// TwinCAT 3 PLC project PLC
// ProgramVersion: 3.1.4024.0
// libraries:
//   SPT Base Types, * (Beckhoff Automation LLC)
//   SPT Components, * (Beckhoff Automation LLC)
//   SPT Diagnostic, * (Beckhoff Automation LLC)
//   SPT EtherCat, * (Beckhoff Automation LLC)
//   SPT Event Logger, * (Beckhoff Automation LLC)
//   SPT Kinematics, * (Beckhoff Automation LLC)
//   SPT Motion Control, * (Beckhoff Automation LLC)
//   SPT NCI, * (Beckhoff Automation LLC)
//   SPT Utilities, * (Beckhoff Automation LLC)
//   SPT Vision, * (Beckhoff Automation LLC)
//   SPT XTS, * (Beckhoff Automation LLC)
//   Tc2_MC2, * (Beckhoff Automation GmbH)
//   Tc2_Standard, * (Beckhoff Automation GmbH)
//   Tc2_System, * (Beckhoff Automation GmbH)
//   Tc3_EventLogger, * (Beckhoff Automation GmbH)
//   Tc3_Module, * (Beckhoff Automation GmbH)
//   Tc3_PackML_V2, * (Beckhoff Automation GmbH)
// project tree:
//   / FastTask.TcTTO, GlobalTextList.TcGTLO, PlcTask.TcTTO, Visualization Manager.TcVMO (not stored)
//   Function Blocks/ExternalSetpointGenerator/ E_ExternalSPGen.TcDUT, FB_ExternalSetpointGenerator.TcPOU, I_ExternalSetpointGenerator.TcIO
//   Modules/00 Machine/ Machine.TcPOU
//   Modules/01 Infeed Position/ Infeed.TcPOU
//   Modules/02 Outfeed Velocity/ Outfeed.TcPOU
//   POUs Fast Task/ BasicESPG_Position.TcPOU, BasicESPG_Velocity.TcPOU, Fast_Task.TcPOU
//   POUs/ MAIN.TcPOU
//   VISUs/ Visualization.TcVIS, Basic_ESPG.TcVIS
// real-time tasks:
//   TASK PlcTask: cycle T#10ms, priority 20, ADS port 350
//   TASK FastTask: cycle T#2ms, priority 1, ADS port 351
// motion (NC):
//   TASK NC-Task 1 SAF: cycle T#2ms, priority 4, ADS port 501
//   TASK NC-Task 1 SVB: cycle T#10ms, priority 8, ADS port 511
//   AXIS Axis Position (id 1)
//     OtherSettings: AllowMotionCmdToSlave=true
//     encoder EncType=1
//     drive DrvType=5
//       Analog: TorqueSetpointScale=10, ScaleFactorActTorque=0.1
//       TimeComp: TaskDelayCycles=1
//     controller CtrType=1
//       CtrPara: PriorControlFactor=1
//         Observer: BandWidth=20
//   AXIS Axis Velocity (id 4)
//     OtherSettings: AllowMotionCmdToSlave=true
//     encoder EncType=1
//     drive DrvType=5
//       Analog: TorqueSetpointScale=10, ScaleFactorActTorque=0.1
//       TimeComp: TaskDelayCycles=1
//     controller CtrType=1
//       CtrPara: PriorControlFactor=1
//         Observer: BandWidth=20
//   AXIS Basic ESPG Velocity (id 3)
//   AXIS Basic ESPG Position (id 2)
// variable links:
//   PLC/PLC Instance <-> NC-Task 1 SAF/Axes/Axis Position
//     FastTask Inputs/Fast_Task.PositionAxis.BasicAxis._Axis.NcToPlc <-> Outputs/ToPlc
//     FastTask Outputs/Fast_Task.PositionAxis.BasicAxis._Axis.PlcToNc <-> Inputs/FromPlc
//   PLC/PLC Instance <-> NC-Task 1 SAF/Axes/Axis Velocity
//     FastTask Inputs/Fast_Task.VelocityAxis.BasicAxis._Axis.NcToPlc <-> Outputs/ToPlc
//     FastTask Outputs/Fast_Task.VelocityAxis.BasicAxis._Axis.PlcToNc <-> Inputs/FromPlc
//   PLC/PLC Instance <-> NC-Task 1 SAF/Axes/Basic ESPG Position
//     FastTask Inputs/BasicESPG_Position.Basic_Axis.NcToPlc <-> Outputs/ToPlc
//     FastTask Outputs/BasicESPG_Position.Basic_Axis.PlcToNc <-> Inputs/FromPlc
//   PLC/PLC Instance <-> NC-Task 1 SAF/Axes/Basic ESPG Velocity
//     FastTask Inputs/BasicESPG_Velocity.Basic_Axis.NcToPlc <-> Outputs/ToPlc
//     FastTask Outputs/BasicESPG_Velocity.Basic_Axis.PlcToNc <-> Inputs/FromPlc

CONFIGURATION PLC
    RESOURCE PLC ON TwinCAT3
        TASK FastTask(INTERVAL := T#2ms, PRIORITY := 1);
        TASK PlcTask(INTERVAL := T#10ms, PRIORITY := 20);
        PROGRAM Fast_Task WITH FastTask : Fast_Task;
        PROGRAM MAIN WITH PlcTask : MAIN;
    END_RESOURCE
END_CONFIGURATION

// ---- Function Blocks/ExternalSetpointGenerator/E_ExternalSPGen.TcDUT
{attribute 'qualified_only'}
{attribute 'strict'}
TYPE E_ExternalSPGen : (
		Wait := 0,
		EnableCmd,
		Enabling,
		Feeding,
		DisableCmd,
		Disabling,
		Error
	);
END_TYPE

// ---- Function Blocks/ExternalSetpointGenerator/I_ExternalSetpointGenerator.TcIO
INTERFACE I_ExternalSetpointGenerator

PROPERTY Accel : lreal
GET
END_GET
SET
END_SET
END_PROPERTY

PROPERTY Destination : lreal
GET
END_GET
SET
END_SET
END_PROPERTY

PROPERTY Direction : DINT // -1 = negative direction, 0 = standstill, 1 = positive direction
GET
END_GET
SET
END_SET
END_PROPERTY

METHOD Disable : bool
VAR_INPUT
END_VAR
END_METHOD

PROPERTY Position : lreal
GET
END_GET
SET
END_SET
END_PROPERTY

PROPERTY Velocity : lreal
GET
END_GET
SET
END_SET
END_PROPERTY

END_INTERFACE

// ---- POUs Fast Task/Fast_Task.TcPOU
PROGRAM Fast_Task
VAR
	PositionAxis	  : FB_Component_BasicAxis := (Name := 'Position Axis');
	PosExtSetpointGen : FB_ExternalSetpointGenerator;
	VelocityAxis	  : FB_Component_BasicAxis := (Name := 'Velocity Axis');
	VelExtSetpointGen : FB_ExternalSetpointGenerator;
END_VAR

(*
	External Setpoint Generator
	This code is the standard implementation of the External Setpoint Generator
	Use this along with the Bassic_ESPG Visu to become familiar with how it works if you have not used the External Setpoint Generator before
	This code is not used by the SPT Framework Implmentation
*)
BasicESPG_Position();
BasicESPG_Velocity();

(*****************************************************************************************************************************************************************)

(*****************************************************************************************************************************************************************)

(*****************************************************************************************************************************************************************)

(*
	These components are defined in this fast task in order for the values of the External Setpoint Generator
	to be updated and transfered to the motion controler at the speed of the fast task.
	These components are controlled and monitored through their interfaces from an EM 
*)

// Infeed EM
PositionAxis.CyclicLogic();
PositionAxis.ExternalSequence := PosExtSetpointGen;

//Outfeed EM
VelocityAxis.CyclicLogic();
VelocityAxis.ExternalSequence := VelExtSetpointGen;

END_PROGRAM

// ---- Function Blocks/ExternalSetpointGenerator/FB_ExternalSetpointGenerator.TcPOU
FUNCTION_BLOCK FB_ExternalSetpointGenerator EXTENDS FB_CyclicFB IMPLEMENTS I_MotionSequence, I_ExternalSetpointGenerator
VAR
	//Properties
	_Axis		 : I_BasicAxis;
	_Position	 : LREAL;
	_Destination : LREAL := 0.0;
	_Velocity	 : LREAL := 0.0;
	_Accel		 : LREAL := 0.0;
	_Direction	 : DINT	 := 1;

	// FBs
	EnableExtSP	 : MC_ExtSetPointGenEnable;
	DisableExtSP : MC_ExtSetPointGenDisable;

	//Internal Vars
	SequenceStep : INT;
	Options		 : ST_ExtSetPointEnableOptions;
END_VAR

PROPERTY Accel : lreal
GET
Accel := _Accel;
END_GET
SET
_Accel := Accel;
END_SET
END_PROPERTY

{warning 'add property implementation'}
PROPERTY Axis : SPT_Motion_Control.I_BasicAxis
GET
Axis := _Axis;
END_GET
SET
_Axis := Axis;
END_SET
END_PROPERTY

{warning 'add method implementation '}
METHOD CyclicLogic

VAR
	_Pos		 : LREAL;
END_VAR
CASE SequenceStep OF
	E_ExternalSPGen.Wait:
		EnableExtSP(Axis := _Axis.Axis, Execute := FALSE, Position := _Axis.ActualPosition);
		DisableExtSP(Axis := _Axis.Axis, Execute := FALSE);

	E_ExternalSPGen.EnableCmd:
		EnableExtSP(Axis		 := _Axis.Axis,
					Execute		 := TRUE,
					Position	 := _Destination, // Used for Position Monitoring
					PositionType := E_PositionType.POSITIONTYPE_ABSOLUTE,
					Options		 := Options);

		IF EnableExtSP.Enabled THEN
			SequenceStep := E_ExternalSPGen.Feeding;
		END_IF

	E_ExternalSPGen.Feeding:
		MC_ExtSetPointGenFeed(Axis		   := _Axis.Axis,
							  Position	   := _Position,
							  Velocity	   := _Velocity,
							  Acceleration := _Accel,
							  Direction	   := _Direction);

	E_ExternalSPGen.DisableCmd:
		DisableExtSP(Axis := _Axis.Axis, Execute := TRUE);
		SequenceStep := E_ExternalSPGen.Disabling;

	E_ExternalSPGen.Disabling:
		DisableExtSP(Axis := _Axis.Axis, Execute := FALSE);
		IF NOT DisableExtSP.Busy AND NOT DisableExtSP.Enabled THEN
			IF NOT DisableExtSP.Error THEN
				SequenceStep := E_ExternalSPGen.Wait;
			ELSE
				_ErrorID	 := DisableExtSP.ErrorID;
				SequenceStep := E_ExternalSPGen.Error;
			END_IF
		END_IF

	E_ExternalSPGen.Error:
		_Error := TRUE;
END_CASE

IF _Axis.Error THEN
	SequenceStep := E_ExternalSPGen.DisableCmd;
END_IF

//
_Busy := (SequenceStep <> 0) AND (NOT _Axis.Error);
END_METHOD

PROPERTY Destination : lreal
GET
Destination := _Destination;
END_GET
SET
_Destination := Destination;
END_SET
END_PROPERTY

PROPERTY Direction : DINT // -1 = negative direction, 0 = standstill, 1 = positive direction
GET
Direction := _Direction;
END_GET
SET
_Direction := Direction;
END_SET
END_PROPERTY

METHOD Disable : bool
VAR_INPUT
END_VAR
IF (_Axis = 0) THEN
	RETURN;
END_IF

_Busy		 := TRUE;
_Error		 := FALSE;
_ErrorID	 := 0;
SequenceStep := E_ExternalSPGen.DisableCmd;
Disable		 := TRUE;
END_METHOD

{warning 'add method implementation '}
METHOD Execute : BOOL
IF (_Axis = 0) OR _Busy THEN
	RETURN;
END_IF

_Busy		 := TRUE;
_Error		 := FALSE;
_ErrorID	 := 0;
SequenceStep := E_ExternalSPGen.EnableCmd;
Execute		 := TRUE;
END_METHOD

PROPERTY Position : lreal
GET
Position := _Position;
END_GET
SET
_Position := Position;
END_SET
END_PROPERTY

PROPERTY Velocity : lreal
GET
Velocity := _Velocity;
END_GET
SET
_Velocity := Velocity;
END_SET
END_PROPERTY

END_FUNCTION_BLOCK

// ---- POUs Fast Task/BasicESPG_Position.TcPOU
PROGRAM BasicESPG_Position
VAR
	Basic_Axis : AXIS_REF;
	Power	   : MC_Power;
	EnableSPG  : MC_ExtSetPointGenEnable;
	DisableSPG : MC_ExtSetPointGenDisable;

	//
	Execute					: BOOL;
	Destination				: LREAL;
	NextIncrementalPosition : LREAL;
	
	Inc1: BOOL;
	Inc10: BOOL;
	Dec1: BOOL;
	Dec10: BOOL;
	HasJob: BOOL;
END_VAR

// The Axis is always enabled for demo purposes
Power(Axis			  := Basic_Axis,
	  Enable		  := TRUE,
	  Enable_Positive := TRUE,
	  Enable_Negative := TRUE);

(*
	Enable the External Setpoint Generator and set the Destination
	The Destination value is loaded when the ESPG is ENabled
	This value will be used to determine the 'In Target Pos' and 'In Pos Range' flags
*)
EnableSPG(Axis := Basic_Axis, Execute := Execute, Position := Destination);

// Disable the External Setpoint Generator when not enabled
DisableSPG(Axis := Basic_Axis, Execute := NOT Execute);

(*
	Once enabled above, the Position value can be modified to send commands to the axis through the Axis.PlcToNc.ExtSetPos
	Velocity is not required as the MC_ExtSetPointGenFeed is sending position commands to the axis 
	- Actualy velocity for a real axis will be based on encoder feedback
	- For a simulation axis, actual velocity will be calculated based on the change in position and the task time
	An Acceleration value is not required for Position commands
	If the Direction is 0 the axis will not move, set the value to 1 for movemnt. The actual direction will be determined by the change in Position
*)

// When the Axis Status 'Has Job' is true, no other commands can be sent to the Axis. While the ESPG is Enabled, the 'Has Job' will be TRUE 
HasJob := Basic_Axis.NcToPlc.StateDWord.8;

//
IF EnableSPG.Enabled THEN // Not required, but prevents the NextIncrementalPosition value from being sent to Axis.PlcToNc.ExtSetPos
	MC_ExtSetPointGenFeed(Axis		   := Basic_Axis,
						  Position	   := NextIncrementalPosition,
						  Velocity	   := 0,
						  Acceleration := 0,
						  Direction	   := 1);
END_IF

(*	WARNING !!!!!!!!
	Changing the Position while the ESPG is not Enabled will change the value of the Axis.PlcToNc.ExtSetPos, but will not cause Axis movement.
	Enabling the ESPG with a Position value that is different than the current Actual Value will cause the axis to jump and likely fault.
*)

// Commands from Visu
IF Inc1 THEN
	Inc1					:= FALSE;
	NextIncrementalPosition := NextIncrementalPosition + 1;
END_IF

IF Inc10 THEN
	Inc10					:= FALSE;
	NextIncrementalPosition := NextIncrementalPosition + 10;
END_IF

IF Dec1 THEN
	Dec1					:= FALSE;
	NextIncrementalPosition := NextIncrementalPosition - 1;
END_IF

IF Dec10 THEN
	Dec10					:= FALSE;
	NextIncrementalPosition := NextIncrementalPosition - 10;
END_IF

END_PROGRAM

// ---- POUs Fast Task/BasicESPG_Velocity.TcPOU
PROGRAM BasicESPG_Velocity
VAR
	Basic_Axis : AXIS_REF;
	Power	   : MC_Power;
	EnableSPG  : MC_ExtSetPointGenEnable;
	DisableSPG : MC_ExtSetPointGenDisable;

	//
	Execute					: BOOL;
	NextIncrementalVelocity : LREAL;
	
	Inc1: BOOL;
	Inc10: BOOL;
	Dec1: BOOL;
	Dec10: BOOL;
	HasJob: BOOL;
END_VAR

// The Axis is always enabled for demo purposes
Power(Axis			  := Basic_Axis,
	  Enable		  := TRUE,
	  Enable_Positive := TRUE,
	  Enable_Negative := TRUE);

// Enable the External Setpoint Generator
EnableSPG(Axis := Basic_Axis, Execute := Execute, Position := 0);

// Disable the External Setpoint Generator when not enabled
DisableSPG(Axis := Basic_Axis, Execute := NOT Execute);

(*
	Once enabled above, the Velocity value can be modified to send commands to the axis through the Axis.PlcToNc.ExtSetVelo
	Position is not required as the MC_ExtSetPointGenFeed is sending Velocity commands to the axis 
	- Actualy velocity for a real axis will be based on encoder feedback
	- For a simulation axis, actual velocity will be 0 and the Actual Position will not change
	An Acceleration value is not required for Velocity commands
	If the Direction is 0 the axis will not move, set the value to 1 for movemnt. The actual direction will be determined by the sign of the Velocity
*)

// When the Axis Status 'Has Job' is true, no other commands can be sent to the Axis. While the ESPG is Enabled, the 'Has Job' will be TRUE 
HasJob := Basic_Axis.NcToPlc.StateDWord.8;

//
IF EnableSPG.Enabled THEN // Not required, but prevents the NextIncrementalVelocity value from being sent to Axis.PlcToNc.ExtSetVelo
	MC_ExtSetPointGenFeed(Axis		   := Basic_Axis,
						  Position	   := 0,
						  Velocity	   := NextIncrementalVelocity,
						  Acceleration := 0,
						  Direction	   := 1);
END_IF

(*	WARNING !!!!!!!!
	Changing the Velocity while the ESPG is not Enabled will change the value of the Axis.PlcToNc.ExtSetVelo, but will not cause Axis movement.
*)

// Commands from Visu
IF Inc1 THEN
	Inc1					:= FALSE;
	NextIncrementalVelocity := NextIncrementalVelocity + 1;
END_IF

IF Inc10 THEN
	Inc10					:= FALSE;
	NextIncrementalVelocity := NextIncrementalVelocity + 10;
END_IF

IF Dec1 THEN
	Dec1					:= FALSE;
	NextIncrementalVelocity := NextIncrementalVelocity - 1;
END_IF

IF Dec10 THEN
	Dec10					:= FALSE;
	NextIncrementalVelocity := NextIncrementalVelocity - 10;
END_IF

END_PROGRAM

// ---- POUs/MAIN.TcPOU
PROGRAM MAIN
VAR
	Machine : Machine := (Name := 'Machine');
END_VAR

(*All sample code provided by Beckhoff Automation LLC are for illustrative purposes only and are provided “as is” and without any warranties, express or implied. Actual implementations in applications will vary significantly. Beckhoff Automation LLC shall have no liability for, and does not waive any rights in relation to, any code samples that it provides or the use of such code samples for any purpose.*)

// NOTE: This code has not been tested on Hardware

// This is for debug only and should be removed
_AppInfo.KeepOutputsOnBP := TRUE;

(*
	There are 2 Equipment modules that use 1 axis each
	The Infeed EM controls an axis that implements Position control
	The Outfeed EM controls an axis that implements Velocity control
	
	Because the External Setpoint Generator provides smoother performce in a faster task,
	the Axis Components are defined within a POU that is updated by a 2ms Fast_Task.

	The fast task only calls the cyclic logic of the components, and sets the External Sequence of the component to the External Setpoint Generator.
	The EMs defined under the Machine Module have an interface that is assigned to the components in the Fast_Task.
	Through this interface the EM can control the component as if it was defined locally.
*)
Machine.CyclicLogic();

END_PROGRAM

// ---- Modules/00 Machine/Machine.TcPOU
FUNCTION_BLOCK Machine EXTENDS FB_PackML_BaseModule
VAR
	Infeed	: Infeed  := (Name := 'Infeed');
	Outfeed : Outfeed := (Name := 'Outfeed');
END_VAR

// Automatically enables and disables HMI control based on the PackML mode
METHOD PROTECTED HMIPermissions

// This method is called cyclically by CyclicLogic()
AllowHMIControl(TRUE);
END_METHOD

// Basic module initialization logic
METHOD PROTECTED Initialize : BOOL;
VAR
END_VAR

// This method is called by CyclicLogic() as required
Initialize := FALSE;
CASE DescendantSequenceState OF
	0:
		RegisterSubmodule(SubModule := Infeed);
		RegisterSubmodule(SubModule := Outfeed);
		DescendantSequenceState := DescendantSequenceState + 10;

	10:
		IF SUPER^.Initialize() THEN
			DescendantSequenceState := DescendantSequenceState + 10;
		END_IF

	20:
		Initialize := TRUE;
END_CASE
END_METHOD

END_FUNCTION_BLOCK

// ---- Modules/01 Infeed Position/Infeed.TcPOU
FUNCTION_BLOCK Infeed EXTENDS FB_PackML_BaseModule
VAR
	iInfeedxis				   : I_BasicAxis;				  // For most axis and component commands
	iInfeedAxisComponent	   : I_ComponentBase;			  // For registering the component with the EM
	iExternalSetpointGenerator : I_ExternalSetpointGenerator; // For setting properties of the External Setpoint Generator
END_VAR

// This method contains code which will execute when this PackML module is in the Aborting state
METHOD PROTECTED Aborting
VAR
	i				: UDINT;
	SubModulesReady : BOOL := TRUE;
END_VAR

// Note: The Abort command should be associated with the fault handing routine of a module. It should not be directly commanded from any user inteface. 

// This method is called as required by <c>StateControl()</c>
CASE SequenceState OF
	0:
		NoStateTasksToComplete := FALSE;
		SequenceState		   := SequenceState + 10;

	10:
		IF NOT iInfeedxis.Error THEN
			IF iInfeedxis.Stop() THEN
				SequenceState := SequenceState + 10;
			END_IF
		ELSE
			SequenceState := SequenceState + 10;
		END_IF

	20:
		IF iInfeedxis.Stopped THEN
			SequenceState := SequenceState + 10;
		END_IF

	30:
		IF iInfeedxis.Disable() THEN
			SequenceState := SequenceState + 10;
		END_IF

	40:
		IF NOT iInfeedxis.Enabled THEN
			SequenceState := SequenceState + 10;
		END_IF

	50:
		StateTasksComplete := TRUE;
END_CASE

SUPER^.Aborting();
END_METHOD

// This method contains code which will execute when this PackML module is in the Clearing state
METHOD PROTECTED Clearing
VAR
	i				: UDINT;
	SubModulesReady : BOOL := TRUE;
END_VAR

// Note: The Clear command can also be thought of as a fault reset depite the ambiguity in the naming of the Reset state. 

// This method is called as required by <c>StateControl()</c>
CASE SequenceState OF
	0:
		NoStateTasksToComplete := FALSE;
		SequenceState		   := SequenceState + 10;

	10:
		IF iInfeedxis.Reset() THEN
			SequenceState := SequenceState + 10;
		END_IF

	20:
		IF NOT iInfeedxis.Error THEN
			SequenceState := SequenceState + 10;
		END_IF

	30:
		StateTasksComplete := TRUE;
END_CASE

SUPER^.Clearing();
END_METHOD

// This method contains code which will execute when this PackML module is in the Execute state
METHOD PROTECTED Execute

(*
The base implementation of this method is empty. User must override this method to provide functionality.
This method is called as required by StateControl()
*)

VAR
	Position: LREAL;
END_VAR
CASE _CurrentMode OF
	E_PMLUnitMode.ePMLUnitMode_Production:
		CASE SequenceState OF
			0:
				iExternalSetpointGenerator.Direction   := 1;
				iExternalSetpointGenerator.Destination := 100.0;
				iExternalSetpointGenerator.Velocity	   := 0.0;
				iExternalSetpointGenerator.Accel	   := 0.0;
				SequenceState						   := 10;

			10:
				IF iInfeedxis.RunExternalSequence() THEN
					SequenceState := 20;
				END_IF

			20:
				IF iInfeedxis.Axis.Status.HasJob THEN //Setpoint generator is operational
					SequenceState := 30;
				END_IF

			30: // Move from 0 to Destination
				Position := iInfeedxis.ActualPosition + ((iExternalSetpointGenerator.Destination - iInfeedxis.ActualPosition) * 0.01);

				iExternalSetpointGenerator.Position := Position;
				IF iInfeedxis.InPosition THEN
					SequenceState := 40;
				END_IF

			40:
				IF iExternalSetpointGenerator.Disable() THEN
					SequenceState := 50;
				END_IF

			50:
				;
		END_CASE
END_CASE
END_METHOD

// Basic module initialization logic
METHOD PROTECTED Initialize : BOOL;
VAR
END_VAR

// This method is called by CyclicLogic() as required
Initialize := FALSE;
CASE DescendantSequenceState OF
	0:
		// Interfaces to connect to Components in the Fast_Task
		iInfeedxis				   := Fast_Task.PositionAxis;	   // For most axis and component commands
		iInfeedAxisComponent	   := Fast_Task.PositionAxis;	   // For registering the component with the EM
		iExternalSetpointGenerator := Fast_Task.PosExtSetpointGen; // For setting properties of the External Setpoint Generator

		//
		RegisterComponent(Component := iInfeedAxisComponent);
		DescendantSequenceState := DescendantSequenceState + 10;

	10:
		IF SUPER^.Initialize() THEN
			DescendantSequenceState := DescendantSequenceState + 10;
		END_IF

	20:
		Initialize := TRUE;
END_CASE
END_METHOD

METHOD PROTECTED Resetting
VAR
END_VAR
CASE SequenceState OF
	0:
		NoStateTasksToComplete := FALSE;
		SequenceState		   := SequenceState + 10;

	10:
		IF iInfeedxis.Enable() THEN
			SequenceState := SequenceState + 10;
		END_IF

	20:
		IF iInfeedxis.Enabled THEN
			SequenceState := SequenceState + 10;
		END_IF

	30:
		StateTasksComplete := TRUE;
END_CASE

SUPER^.Resetting();
END_METHOD

END_FUNCTION_BLOCK

// ---- Modules/02 Outfeed Velocity/Outfeed.TcPOU
FUNCTION_BLOCK Outfeed EXTENDS FB_PackML_BaseModule
VAR
	iOutfeedxis				   : I_BasicAxis;				  // For most axis and component commands
	iOutfeedAxisComponent	   : I_ComponentBase;			  // For registering the component with the EM
	iExternalSetpointGenerator : I_ExternalSetpointGenerator; // For setting properties of the External Setpoint Generator
END_VAR

// This method contains code which will execute when this PackML module is in the Aborting state
METHOD PROTECTED Aborting

// Note: The Abort command should be associated with the fault handing routine of a module. It should not be directly commanded from any user inteface. 

// This method is called as required by <c>StateControl()</c>
CASE SequenceState OF
	0:
		NoStateTasksToComplete := FALSE;
		SequenceState		   := SequenceState + 10;

	10:
		IF NOT iOutfeedxis.Error THEN
			IF iOutfeedxis.Stop() THEN
				SequenceState := SequenceState + 10;
			END_IF
		ELSE
			SequenceState := SequenceState + 10;
		END_IF

	20:
		IF iOutfeedxis.Stopped THEN
			SequenceState := SequenceState + 10;
		END_IF

	30:
		IF iOutfeedxis.Disable() THEN
			SequenceState := SequenceState + 10;
		END_IF

	40:
		IF NOT iOutfeedxis.Enabled THEN
			SequenceState := SequenceState + 10;
		END_IF

	50:
		StateTasksComplete := TRUE;
END_CASE

SUPER^.Aborting();
END_METHOD

// This method contains code which will execute when this PackML module is in the Clearing state
METHOD PROTECTED Clearing
VAR
	i				: UDINT;
	SubModulesReady : BOOL := TRUE;
END_VAR

// Note: The Clear command can also be thought of as a fault reset depite the ambiguity in the naming of the Reset state. 

// This method is called as required by <c>StateControl()</c>
CASE SequenceState OF
	0:
		NoStateTasksToComplete := FALSE;
		SequenceState		   := SequenceState + 10;

	10:
		IF iOutfeedxis.Reset() THEN
			SequenceState := SequenceState + 10;
		END_IF

	20:
		IF NOT iOutfeedxis.Error THEN
			SequenceState := SequenceState + 10;
		END_IF

	30:
		StateTasksComplete := TRUE;
END_CASE

SUPER^.Clearing();
END_METHOD

// This method contains code which will execute when this PackML module is in the Execute state
METHOD PROTECTED Execute
VAR
	

END_VAR

(*
The base implementation of this method is empty. User must override this method to provide functionality.
This method is called as required by StateControl()
*)
VAR
	Position : LREAL;
END_VAR
CASE _CurrentMode OF
	E_PMLUnitMode.ePMLUnitMode_Production:
		CASE SequenceState OF
			0:
				iExternalSetpointGenerator.Direction   := 1;
				iExternalSetpointGenerator.Destination := 0.0;
				iExternalSetpointGenerator.Velocity	   := 0.0;
				iExternalSetpointGenerator.Accel	   := 0.0;
				SequenceState						   := 10;

			10:
				IF iOutfeedxis.RunExternalSequence() THEN
					SequenceState := 20;
				END_IF

			20:
				IF iOutfeedxis.Axis.Status.HasJob THEN //Setpoint generator is operational
					SequenceState := 30;
				END_IF

			30: // Raise Velocity

				//ExtSetpointGen.Velocity := VelocityAxis.ActualVelocity + ((100.0 - VelocityAxis.ActualVelocity) * 0.01); // Without encoder feedback the Actual Velocity will stay at 0
				iExternalSetpointGenerator.Velocity := iExternalSetpointGenerator.Velocity + 0.01;
				IF iOutfeedxis.SetVelocity > 100.0 THEN
					SequenceState := 40;
				END_IF

			40: // Reduce Velocity to 0

				//ExtSetpointGen.Velocity := VelocityAxis.ActualVelocity - ((0.0 - VelocityAxis.ActualVelocity) * 0.01); // Without encoder feedback the Actual Velocity will stay at 0
				iExternalSetpointGenerator.Velocity := iExternalSetpointGenerator.Velocity - 0.01;
				IF (iExternalSetpointGenerator.Velocity <= 1.0) AND (iOutfeedxis.ActualVelocity = 0) THEN
					SequenceState := 50;
				END_IF

			50:
				IF iExternalSetpointGenerator.Disable() THEN
					SequenceState := 60;
				END_IF

			60:
				;
		END_CASE
END_CASE
END_METHOD

// Basic module initialization logic
METHOD PROTECTED Initialize : BOOL;
VAR
END_VAR

// This method is called by CyclicLogic() as required
Initialize := FALSE;
CASE DescendantSequenceState OF
	0:
		// Interfaces to connect to Components in the Fast_Task
		iOutfeedxis				   := Fast_Task.VelocityAxis;	   // For most axis and component commands
		iOutfeedAxisComponent	   := Fast_Task.VelocityAxis;	   // For registering the component with the EM
		iExternalSetpointGenerator := Fast_Task.VelExtSetpointGen; // For setting properties of the External Setpoint Generator

		//
		RegisterComponent(Component := iOutfeedAxisComponent);
		DescendantSequenceState := DescendantSequenceState + 10;

	10:
		IF SUPER^.Initialize() THEN
			DescendantSequenceState := DescendantSequenceState + 10;
		END_IF

	20:
		Initialize := TRUE;
END_CASE
END_METHOD

METHOD PROTECTED Resetting
VAR
END_VAR
CASE SequenceState OF
	0:
		NoStateTasksToComplete := FALSE;
		SequenceState		   := SequenceState + 10;

	10:
		IF iOutfeedxis.Enable() THEN
			SequenceState := SequenceState + 10;
		END_IF

	20:
		IF iOutfeedxis.Enabled THEN
			SequenceState := SequenceState + 10;
		END_IF

	30:
		StateTasksComplete := TRUE;
END_CASE

SUPER^.Resetting();
END_METHOD

END_FUNCTION_BLOCK

// ---- GlobalTextList.TcGTLO
TEXTLIST GlobalTextList
  155 = '<'
  625 = '<<'
  160 = '>'
  854 = '>>'
  636 = 'Enable SPG'
  612 = 'ExtSetPos: %2.5f'
  338 = 'ExtSetPos: %5.2f'
  808 = 'ExtSetPos: %f'
  435 = 'ExtSetVelo: %f'
  81 = 'Set Position Value: %5.2f'
  13 = 'Set Position Value: %f'
  748 = 'Set Velocity Value: %5.2f'
END_TEXTLIST

// ---- VISUs/Visualization.TcVIS
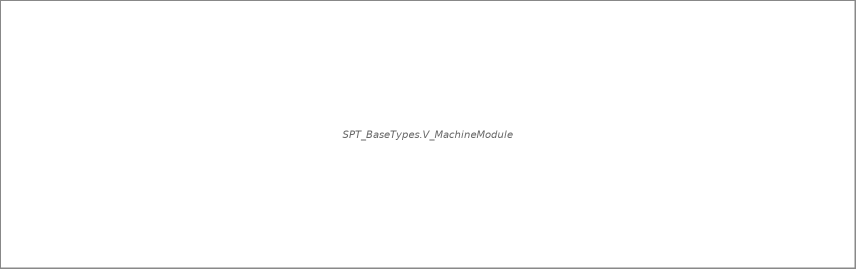
VISUALIZATION Visualization  // 856x269
    Frame (0,0 856x269)
        shows SPT_BaseTypes.V_MachineModule(HMI := MAIN.Machine.PackMLBaseModule_HMI)
END_VISUALIZATION

// ---- VISUs/Basic_ESPG.TcVIS
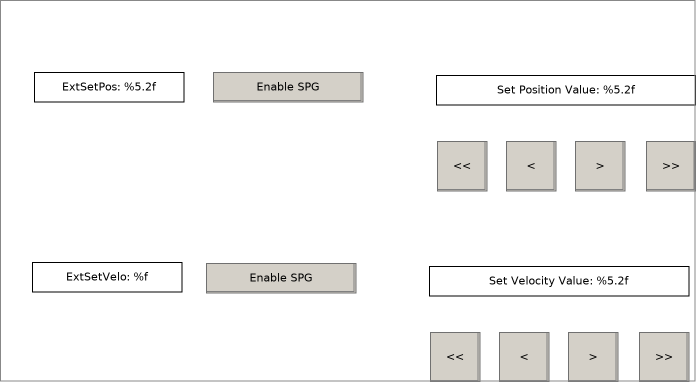
VISUALIZATION Basic_ESPG  // 696x382
    Rectangle (34,72 150x30), "ExtSetPos: %5.2f", text variable: BasicESPG_Position.Basic_Axis.PlcToNc.ExtSetPos
    Rectangle (32,262 150x30), "ExtSetVelo: %f", text variable: BasicESPG_Velocity.Basic_Axis.PlcToNc.ExtSetVelo
    Button (213,72 150x30), "Enable SPG"
        toggle BasicESPG_Position.Execute
    Rectangle (436,75 260x30), "Set Position Value: %5.2f", text variable: BasicESPG_Position.NextIncrementalPosition
    Button (575,141 50x50), ">"
        toggle BasicESPG_Position.Inc1
    Button (646,141 50x50), ">>"
        toggle BasicESPG_Position.Inc10
    Button (506,141 50x50), "<"
        toggle BasicESPG_Position.Dec1
    Button (437,141 50x50), "<<"
        toggle BasicESPG_Position.Dec10
    Button (206,263 150x30), "Enable SPG"
        toggle BasicESPG_Velocity.Execute
    Rectangle (429,266 260x30), "Set Velocity Value: %5.2f", text variable: BasicESPG_Velocity.NextIncrementalVelocity
    Button (568,332 50x50), ">"
        toggle BasicESPG_Velocity.Inc1
    Button (639,332 50x50), ">>"
        toggle BasicESPG_Velocity.Inc10
    Button (499,332 50x50), "<"
        toggle BasicESPG_Velocity.Dec1
    Button (430,332 50x50), "<<"
        toggle BasicESPG_Velocity.Dec10
END_VISUALIZATION
